Universal Robots PolyScope program: annaetest2.urp

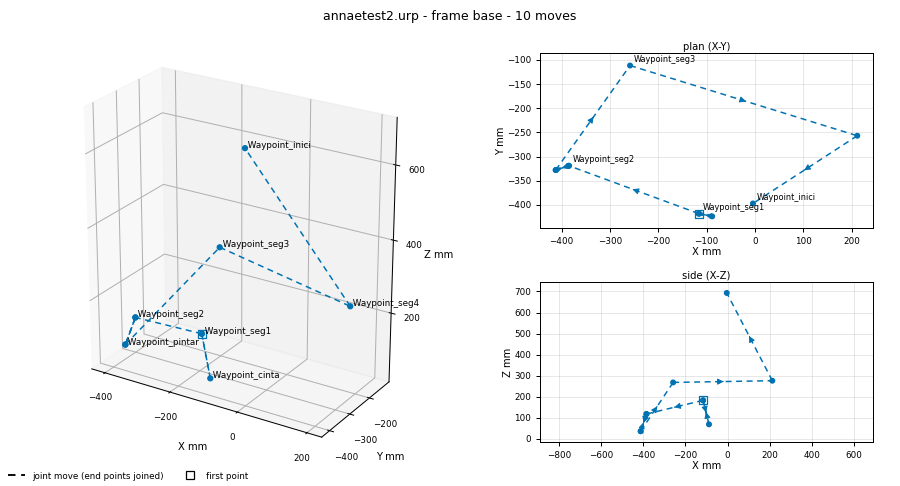
[picture p0: tool path of annaetest2.urp in frame base, 10 of 10 moves have a stored position in this frame; points joined in program order, loops and branches not executed]
Program annaetest2 (installation=default directory=/programs createdIn=5.14.5 lastSavedIn=5.14.5 robotSerialNumber=20195300809)
Calibrated DH parameters: a=[-0.000085, -0.20076, -0.212369, 0.000121, -0.000118, 0]; d=[0.15185, -26.306375, 24.753047, 1.684739, 0.085386, 0.092088]; alpha=[1.572149, -0.00522, -0.011864, 1.571339, -1.571085, 0]; deltaTheta=[0, 0.599885, -0.513355, -0.086555, 0.000006, 0]
InitVariablesNode
BeforeStart
  finished := True
  SafeHome (positionOptionType=SPEED_AND_ACCELERATION speed=1.047198 acceleration=1.396263 nextMotionTime=2)
  Set DigitalOutput pin=digital_out[0]; digitalValue=0
  URCap Gripper Activate (Robotiq_Grippers, Robotiq Inc.) dataModel(ResetAndActivateKey=false)
  URCap Gripper (Robotiq_Grippers, Robotiq Inc.) dataModel(position=0.0, force=0.0, speed=0.0, positionInDouble=0.0, forceInDouble=0.0, speedInDouble=0.0, slaveIds=[9], blocking=true)
Robot Program (runOnlyOnce=false)
  Set DigitalOutput pin=digital_out[0]; digitalValue=1
  If digital_in[0]≟0 (checkContinuously=true)
    Set DigitalOutput pin=digital_out[0]; digitalValue=0
    If finished≟ True (checkContinuously=true)
      finished := False
      MoveJ speed 60 deg/s, acceleration 80 deg/s^2 (useActiveTCP=true) feature=Base
        Waypoint Waypoint_seg1: TCP in base x=-116.459 y=-418.097 z=183.306 mm, rx=0.0468 ry=3.1181 rz=-0.0427 rad; joints [55.479, -57.904, 33.342, -66.043, -88.88, -32.484] deg; TCP offset x=0 y=0 z=174 mm, rx=0 ry=0 rz=0 rad
        Wait Sleep waitTime=1
        MoveJ speed 60 deg/s, acceleration 80 deg/s^2 (useActiveTCP=true) feature=Base
          Waypoint Waypoint_cinta: TCP in base x=-88.455 y=-423.884 z=69.425 mm, rx=0.0423 ry=3.0378 rz=0.0064 rad; joints [57.287, -59.662, 66.287, -93.294, -85.953, -31.25] deg
          URCap Gripper (Robotiq_Grippers, Robotiq Inc.) dataModel(position=100.0, force=0.0, speed=0.0, positionInDouble=100.0, forceInDouble=0.0, speedInDouble=0.0, slaveIds=[9], blocking=true)
          Wait Sleep waitTime=1
          Waypoint Waypoint_seg1: TCP in base x=-116.459 y=-418.097 z=183.306 mm, rx=0.0468 ry=3.1181 rz=-0.0427 rad; joints [55.479, -57.904, 33.342, -66.043, -88.88, -32.484] deg
          Set DigitalOutput pin=digital_out[0]; digitalValue=1
          MoveJ speed 60 deg/s, acceleration 80 deg/s^2 (useActiveTCP=true) feature=Base
            Waypoint Waypoint_seg2: TCP in base x=-385.09 y=-319.115 z=118.622 mm, rx=0.0245 ry=-3.1262 rz=0.0019 rad; joints [24.615, -30.68, 0.967, -61.125, -91.135, -66.065] deg
          MoveJ speed 60 deg/s, acceleration 80 deg/s^2 (useActiveTCP=true) feature=Base
            Waypoint Waypoint_pintar: TCP in base x=-412.438 y=-327.987 z=36.934 mm, rx=0.0644 ry=3.1149 rz=-0.0018 rad; joints [23.765, -20.553, 2.59, -70.73, -90.186, -63.802] deg
          URCap Gripper (Robotiq_Grippers, Robotiq Inc.) dataModel(position=0.0, force=0.0, speed=0.0, positionInDouble=0.0, forceInDouble=0.0, speedInDouble=0.0, slaveIds=[9], blocking=true)
          MoveJ speed 60 deg/s, acceleration 80 deg/s^2 (useActiveTCP=true) feature=Base
            Waypoint Waypoint_seg2: TCP in base x=-385.09 y=-319.115 z=118.622 mm, rx=0.0245 ry=-3.1262 rz=0.0019 rad; joints [24.615, -30.68, 0.967, -61.125, -91.135, -66.065] deg
          MoveJ speed 60 deg/s, acceleration 80 deg/s^2 (useActiveTCP=true) feature=Base
            Waypoint Waypoint_pintar: TCP in base x=-412.438 y=-327.987 z=36.934 mm, rx=0.0644 ry=3.1149 rz=-0.0018 rad; joints [23.765, -20.553, 2.59, -70.73, -90.186, -63.802] deg
          URCap Gripper (Robotiq_Grippers, Robotiq Inc.) dataModel(position=100.0, force=0.0, speed=0.0, positionInDouble=100.0, forceInDouble=0.0, speedInDouble=0.0, slaveIds=[9], blocking=true)
          MoveJ speed 60 deg/s, acceleration 80 deg/s^2 (useActiveTCP=true) feature=Base
            Waypoint Waypoint_seg3: TCP in base x=-258.5 y=-111.618 z=268.321 mm, rx=0.0353 ry=3.114 rz=0.0033 rad; joints [-4.524, -87.218, 46.008, -47.242, -90.863, -92.594] deg
          MoveJ speed 60 deg/s, acceleration 80 deg/s^2 (useActiveTCP=true) feature=Base
            Waypoint Waypoint_seg4: TCP in base x=211.956 y=-257 z=276.441 mm, rx=-2.2529 ry=2.1601 rz=-0.0158 rad; joints [104.982, -71.476, 23.358, -41.799, -89.356, -76.815] deg
          MoveJ speed 60 deg/s, acceleration 80 deg/s^2 (useActiveTCP=true) feature=Base
            Waypoint Waypoint_inici: TCP in base x=-4.073 y=-397.216 z=692.8 mm, rx=0.0312 ry=2.1769 rz=-2.1754 rad; joints [1.86, -87.236, -4.208, -80.341, -1.018, -4.802] deg
          finished := True
